// Code généré automatiquement : NE PAS MODIFIER
FUNCTION CheckDivLInt : LINT
VAR_INPUT
	divisor:LINT;
END_VAR

// Code généré automatiquement : Il s’agit d’une proposition d’implémentation.
{noflow}
IF divisor = 0 THEN
	CheckDivLInt:=1;
ELSE
	CheckDivLInt:=divisor;
END_IF;
{flow}

END_FUNCTION

(* stored: Version 1.1.0.1, ProductVersion 3.1.4024.6
   POU CheckDivLInt: Id {2a223191-eecf-44eb-a897-e691c183bfde}, SpecialFunc CheckDivInt64 *)
